// TIA Portal V16 export
// export: Created 2023-03-29T11:04:38.8533234Z, ExportSetting WithDefaults, DisplayName Totally Integrated Automation Portal, DisplayVersion V16 Update 6, DisplayName TIA Portal Version Control Interface, DisplayVersion V16 Update 2, DisplayName TIA Portal Openness, DisplayVersion V16 Update 6, DisplayName STEP 7 Professional, DisplayVersion V16 Update 6, DisplayName STEP 7 Safety, DisplayVersion V16, DisplayName WinCC Advanced, DisplayVersion V16 Update 6
FUNCTION "Read_MPP04_1_ModbusRTU" : Void   // FC23, LAD
TITLE = Read data from SC100
{ S7_Optimized_Access := 'TRUE' }
AUTHOR : rtecmer
VERSION : 0.1
// Czytanie z SC1000 
// Obsługa protokołu Master Modbus RTU.  Odczyt pomiarów  i status czujnika SC1000
// stored: AutoNumber true, IsIECCheckEnabled false, SetENOAutomatically false, UDAEnableTagReadback false
   VAR_TEMP   // added for the SCL form of the ladder/FBD networks
      _w1 : Bool;
      _w2 : Bool;
   END_VAR
BEGIN

REGION Network 1
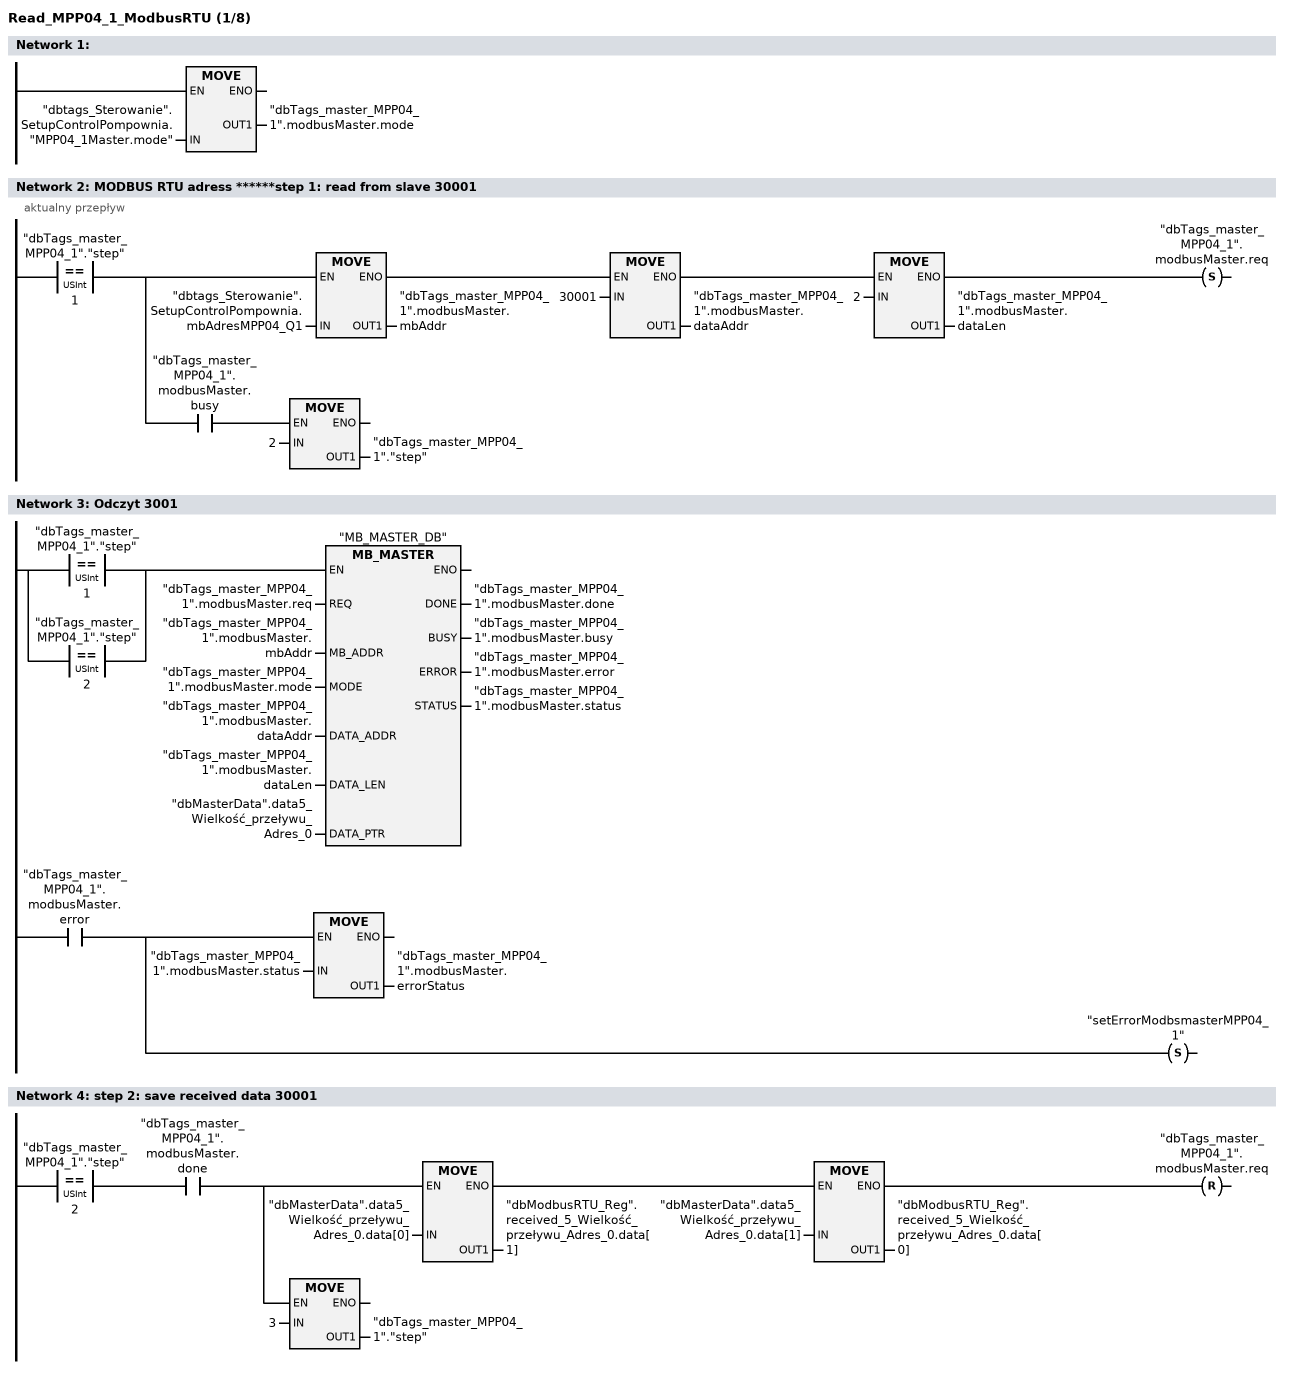
   RUNG wire#powerrail
      { S7_GenerateENO := "TRUE" } Move(in := "dbtags_Sterowanie".SetupControlPompownia."MPP04_1Master.mode", out1 => "dbTags_master_MPP04_1".modbusMaster.mode)
   END_RUNG
   // the same network as SCL:
   "dbTags_master_MPP04_1".modbusMaster.mode := "dbtags_Sterowanie".SetupControlPompownia."MPP04_1Master.mode";
END_REGION

REGION Network 2: MODBUS RTU adress ******step 1: read from slave 30001
   // aktualny przepływ
   RUNG wire#powerrail
      { S7_Templates := "SrcType := USInt" } EQ_Contact(in1 := "dbTags_master_MPP04_1"."step", in2 := 1)
      wire#w1
      Move(in := "dbtags_Sterowanie".SetupControlPompownia.mbAdresMPP04_Q1, out1 => "dbTags_master_MPP04_1".modbusMaster.mbAddr)
      { S7_GenerateENO := "TRUE" } Move(in := 30001, out1 => "dbTags_master_MPP04_1".modbusMaster.dataAddr)
      Move(in := 2, out1 => "dbTags_master_MPP04_1".modbusMaster.dataLen)
      S_Coil( "dbTags_master_MPP04_1".modbusMaster.req )
   END_RUNG
   RUNG wire#w1
      Contact( "dbTags_master_MPP04_1".modbusMaster.busy )
      { S7_GenerateENO := "TRUE" } Move(in := 2, out1 => "dbTags_master_MPP04_1"."step")
   END_RUNG
   // the same network as SCL:
   // ENO of a box is taken as its EN; it also drops when the box reports an error
   #_w1 := "dbTags_master_MPP04_1"."step" = 1;
   IF #_w1 THEN
       "dbTags_master_MPP04_1".modbusMaster.mbAddr := "dbtags_Sterowanie".SetupControlPompownia.mbAdresMPP04_Q1;
       "dbTags_master_MPP04_1".modbusMaster.dataAddr := 30001;
       "dbTags_master_MPP04_1".modbusMaster.dataLen := 2;
       "dbTags_master_MPP04_1".modbusMaster.req := TRUE;
   END_IF;
   IF #_w1 AND "dbTags_master_MPP04_1".modbusMaster.busy THEN "dbTags_master_MPP04_1"."step" := 2; END_IF;
END_REGION

REGION Network 3: Odczyt 3001
   RUNG wire#powerrail
      { S7_Templates := "SrcType := USInt" } EQ_Contact(in1 := "dbTags_master_MPP04_1"."step", in2 := 1)
      wire#w1
      "MB_MASTER_DB".MB_MASTER(REQ := "dbTags_master_MPP04_1".modbusMaster.req, MB_ADDR := "dbTags_master_MPP04_1".modbusMaster.mbAddr, MODE := "dbTags_master_MPP04_1".modbusMaster.mode, DATA_ADDR := "dbTags_master_MPP04_1".modbusMaster.dataAddr, DATA_LEN := "dbTags_master_MPP04_1".modbusMaster.dataLen, DATA_PTR := "dbMasterData".data5_Wielkość_przeływu_Adres_0, DONE => "dbTags_master_MPP04_1".modbusMaster.done, BUSY => "dbTags_master_MPP04_1".modbusMaster.busy, ERROR => "dbTags_master_MPP04_1".modbusMaster.error, STATUS => "dbTags_master_MPP04_1".modbusMaster.status)
   END_RUNG
   RUNG wire#powerrail
      { S7_Templates := "SrcType := USInt" } EQ_Contact(in1 := "dbTags_master_MPP04_1"."step", in2 := 2)
   END_RUNG wire#w1
   RUNG wire#powerrail
      Contact( "dbTags_master_MPP04_1".modbusMaster.error )
      wire#w2
      { S7_GenerateENO := "TRUE" } Move(in := "dbTags_master_MPP04_1".modbusMaster.status, out1 => "dbTags_master_MPP04_1".modbusMaster.errorStatus)
   END_RUNG
   RUNG wire#w2
      S_Coil( "setErrorModbsmasterMPP04_1" )
   END_RUNG
   // the same network as SCL:
   IF ("dbTags_master_MPP04_1"."step" = 1) OR ("dbTags_master_MPP04_1"."step" = 2) THEN
       "MB_MASTER_DB"(REQ := "dbTags_master_MPP04_1".modbusMaster.req,   // MB_MASTER
                      MB_ADDR := "dbTags_master_MPP04_1".modbusMaster.mbAddr,
                      MODE := "dbTags_master_MPP04_1".modbusMaster.mode,
                      DATA_ADDR := "dbTags_master_MPP04_1".modbusMaster.dataAddr,
                      DATA_LEN := "dbTags_master_MPP04_1".modbusMaster.dataLen,
                      DATA_PTR := "dbMasterData".data5_Wielkość_przeływu_Adres_0,
                      DONE => "dbTags_master_MPP04_1".modbusMaster.done,
                      BUSY => "dbTags_master_MPP04_1".modbusMaster.busy,
                      ERROR => "dbTags_master_MPP04_1".modbusMaster.error,
                      STATUS => "dbTags_master_MPP04_1".modbusMaster.status);
   END_IF;
   IF "dbTags_master_MPP04_1".modbusMaster.error THEN
       "dbTags_master_MPP04_1".modbusMaster.errorStatus := "dbTags_master_MPP04_1".modbusMaster.status;
       "setErrorModbsmasterMPP04_1" := TRUE;
   END_IF;
END_REGION

REGION Network 4: step 2: save received data 30001
   RUNG wire#powerrail
      { S7_Templates := "SrcType := USInt" } EQ_Contact(in1 := "dbTags_master_MPP04_1"."step", in2 := 2)
      Contact( "dbTags_master_MPP04_1".modbusMaster.done )
      wire#w1
      { S7_GenerateENO := "TRUE" } Move(in := "dbMasterData".data5_Wielkość_przeływu_Adres_0.data[0], out1 => "dbModbusRTU_Reg".received_5_Wielkość_przeływu_Adres_0.data[1])
      { S7_GenerateENO := "TRUE" } Move(in := "dbMasterData".data5_Wielkość_przeływu_Adres_0.data[1], out1 => "dbModbusRTU_Reg".received_5_Wielkość_przeływu_Adres_0.data[0])
      R_Coil( "dbTags_master_MPP04_1".modbusMaster.req )
   END_RUNG
   RUNG wire#w1
      { S7_GenerateENO := "TRUE" } Move(in := 3, out1 => "dbTags_master_MPP04_1"."step")
   END_RUNG
   // the same network as SCL:
   // ENO of a box is taken as its EN; it also drops when the box reports an error
   IF ("dbTags_master_MPP04_1"."step" = 2) AND "dbTags_master_MPP04_1".modbusMaster.done THEN
       "dbModbusRTU_Reg".received_5_Wielkość_przeływu_Adres_0.data[1] := "dbMasterData".data5_Wielkość_przeływu_Adres_0.data[0];
       "dbModbusRTU_Reg".received_5_Wielkość_przeływu_Adres_0.data[0] := "dbMasterData".data5_Wielkość_przeływu_Adres_0.data[1];
       "dbTags_master_MPP04_1".modbusMaster.req := FALSE;
       "dbTags_master_MPP04_1"."step" := 3;
   END_IF;
END_REGION

REGION Network 5: reakcja na błąd
   // Jęśli błąd pętli modbus lub błąd statusu przepływomierza toustaw 0
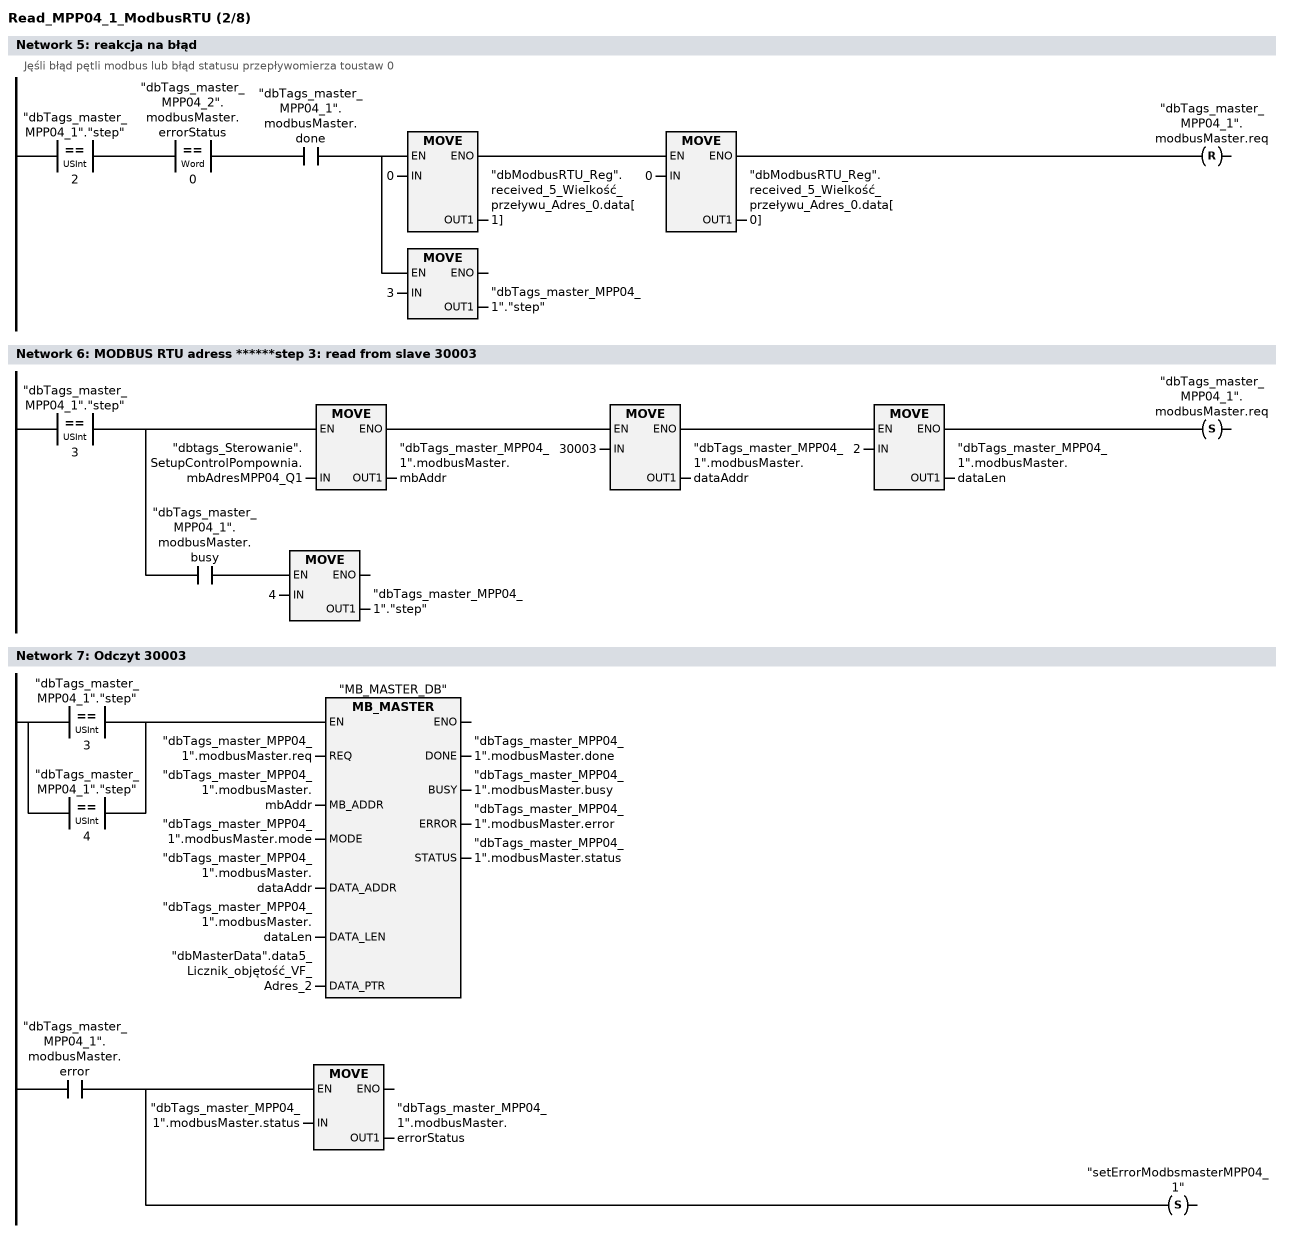
   RUNG wire#powerrail
      { S7_Templates := "SrcType := USInt" } EQ_Contact(in1 := "dbTags_master_MPP04_1"."step", in2 := 2)
      { S7_Templates := "SrcType := Word" } EQ_Contact(in1 := "dbTags_master_MPP04_2".modbusMaster.errorStatus, in2 := 0)
      Contact( "dbTags_master_MPP04_1".modbusMaster.done )
      wire#w1
      { S7_GenerateENO := "TRUE" } Move(in := 0, out1 => "dbModbusRTU_Reg".received_5_Wielkość_przeływu_Adres_0.data[1])
      { S7_GenerateENO := "TRUE" } Move(in := 0, out1 => "dbModbusRTU_Reg".received_5_Wielkość_przeływu_Adres_0.data[0])
      R_Coil( "dbTags_master_MPP04_1".modbusMaster.req )
   END_RUNG
   RUNG wire#w1
      { S7_GenerateENO := "TRUE" } Move(in := 3, out1 => "dbTags_master_MPP04_1"."step")
   END_RUNG
   // the same network as SCL:
   // ENO of a box is taken as its EN; it also drops when the box reports an error
   IF ("dbTags_master_MPP04_1"."step" = 2) AND ("dbTags_master_MPP04_2".modbusMaster.errorStatus = 0) AND "dbTags_master_MPP04_1".modbusMaster.done THEN
       "dbModbusRTU_Reg".received_5_Wielkość_przeływu_Adres_0.data[1] := 0;
       "dbModbusRTU_Reg".received_5_Wielkość_przeływu_Adres_0.data[0] := 0;
       "dbTags_master_MPP04_1".modbusMaster.req := FALSE;
       "dbTags_master_MPP04_1"."step" := 3;
   END_IF;
END_REGION

REGION Network 6: MODBUS RTU adress ******step 3: read from slave 30003
   RUNG wire#powerrail
      { S7_Templates := "SrcType := USInt" } EQ_Contact(in1 := "dbTags_master_MPP04_1"."step", in2 := 3)
      wire#w1
      Move(in := "dbtags_Sterowanie".SetupControlPompownia.mbAdresMPP04_Q1, out1 => "dbTags_master_MPP04_1".modbusMaster.mbAddr)
      { S7_GenerateENO := "TRUE" } Move(in := 30003, out1 => "dbTags_master_MPP04_1".modbusMaster.dataAddr)
      Move(in := 2, out1 => "dbTags_master_MPP04_1".modbusMaster.dataLen)
      S_Coil( "dbTags_master_MPP04_1".modbusMaster.req )
   END_RUNG
   RUNG wire#w1
      Contact( "dbTags_master_MPP04_1".modbusMaster.busy )
      { S7_GenerateENO := "TRUE" } Move(in := 4, out1 => "dbTags_master_MPP04_1"."step")
   END_RUNG
   // the same network as SCL:
   // ENO of a box is taken as its EN; it also drops when the box reports an error
   #_w1 := "dbTags_master_MPP04_1"."step" = 3;
   IF #_w1 THEN
       "dbTags_master_MPP04_1".modbusMaster.mbAddr := "dbtags_Sterowanie".SetupControlPompownia.mbAdresMPP04_Q1;
       "dbTags_master_MPP04_1".modbusMaster.dataAddr := 30003;
       "dbTags_master_MPP04_1".modbusMaster.dataLen := 2;
       "dbTags_master_MPP04_1".modbusMaster.req := TRUE;
   END_IF;
   IF #_w1 AND "dbTags_master_MPP04_1".modbusMaster.busy THEN "dbTags_master_MPP04_1"."step" := 4; END_IF;
END_REGION

REGION Network 7: Odczyt 30003
   RUNG wire#powerrail
      { S7_Templates := "SrcType := USInt" } EQ_Contact(in1 := "dbTags_master_MPP04_1"."step", in2 := 3)
      wire#w1
      "MB_MASTER_DB".MB_MASTER(REQ := "dbTags_master_MPP04_1".modbusMaster.req, MB_ADDR := "dbTags_master_MPP04_1".modbusMaster.mbAddr, MODE := "dbTags_master_MPP04_1".modbusMaster.mode, DATA_ADDR := "dbTags_master_MPP04_1".modbusMaster.dataAddr, DATA_LEN := "dbTags_master_MPP04_1".modbusMaster.dataLen, DATA_PTR := "dbMasterData".data5_Licznik_objętość_VF_Adres_2, DONE => "dbTags_master_MPP04_1".modbusMaster.done, BUSY => "dbTags_master_MPP04_1".modbusMaster.busy, ERROR => "dbTags_master_MPP04_1".modbusMaster.error, STATUS => "dbTags_master_MPP04_1".modbusMaster.status)
   END_RUNG
   RUNG wire#powerrail
      { S7_Templates := "SrcType := USInt" } EQ_Contact(in1 := "dbTags_master_MPP04_1"."step", in2 := 4)
   END_RUNG wire#w1
   RUNG wire#powerrail
      Contact( "dbTags_master_MPP04_1".modbusMaster.error )
      wire#w2
      { S7_GenerateENO := "TRUE" } Move(in := "dbTags_master_MPP04_1".modbusMaster.status, out1 => "dbTags_master_MPP04_1".modbusMaster.errorStatus)
   END_RUNG
   RUNG wire#w2
      S_Coil( "setErrorModbsmasterMPP04_1" )
   END_RUNG
   // the same network as SCL:
   IF ("dbTags_master_MPP04_1"."step" = 3) OR ("dbTags_master_MPP04_1"."step" = 4) THEN
       "MB_MASTER_DB"(REQ := "dbTags_master_MPP04_1".modbusMaster.req,   // MB_MASTER
                      MB_ADDR := "dbTags_master_MPP04_1".modbusMaster.mbAddr,
                      MODE := "dbTags_master_MPP04_1".modbusMaster.mode,
                      DATA_ADDR := "dbTags_master_MPP04_1".modbusMaster.dataAddr,
                      DATA_LEN := "dbTags_master_MPP04_1".modbusMaster.dataLen,
                      DATA_PTR := "dbMasterData".data5_Licznik_objętość_VF_Adres_2,
                      DONE => "dbTags_master_MPP04_1".modbusMaster.done,
                      BUSY => "dbTags_master_MPP04_1".modbusMaster.busy,
                      ERROR => "dbTags_master_MPP04_1".modbusMaster.error,
                      STATUS => "dbTags_master_MPP04_1".modbusMaster.status);
   END_IF;
   IF "dbTags_master_MPP04_1".modbusMaster.error THEN
       "dbTags_master_MPP04_1".modbusMaster.errorStatus := "dbTags_master_MPP04_1".modbusMaster.status;
       "setErrorModbsmasterMPP04_1" := TRUE;
   END_IF;
END_REGION

REGION Network 8: step 4: save received data 30003
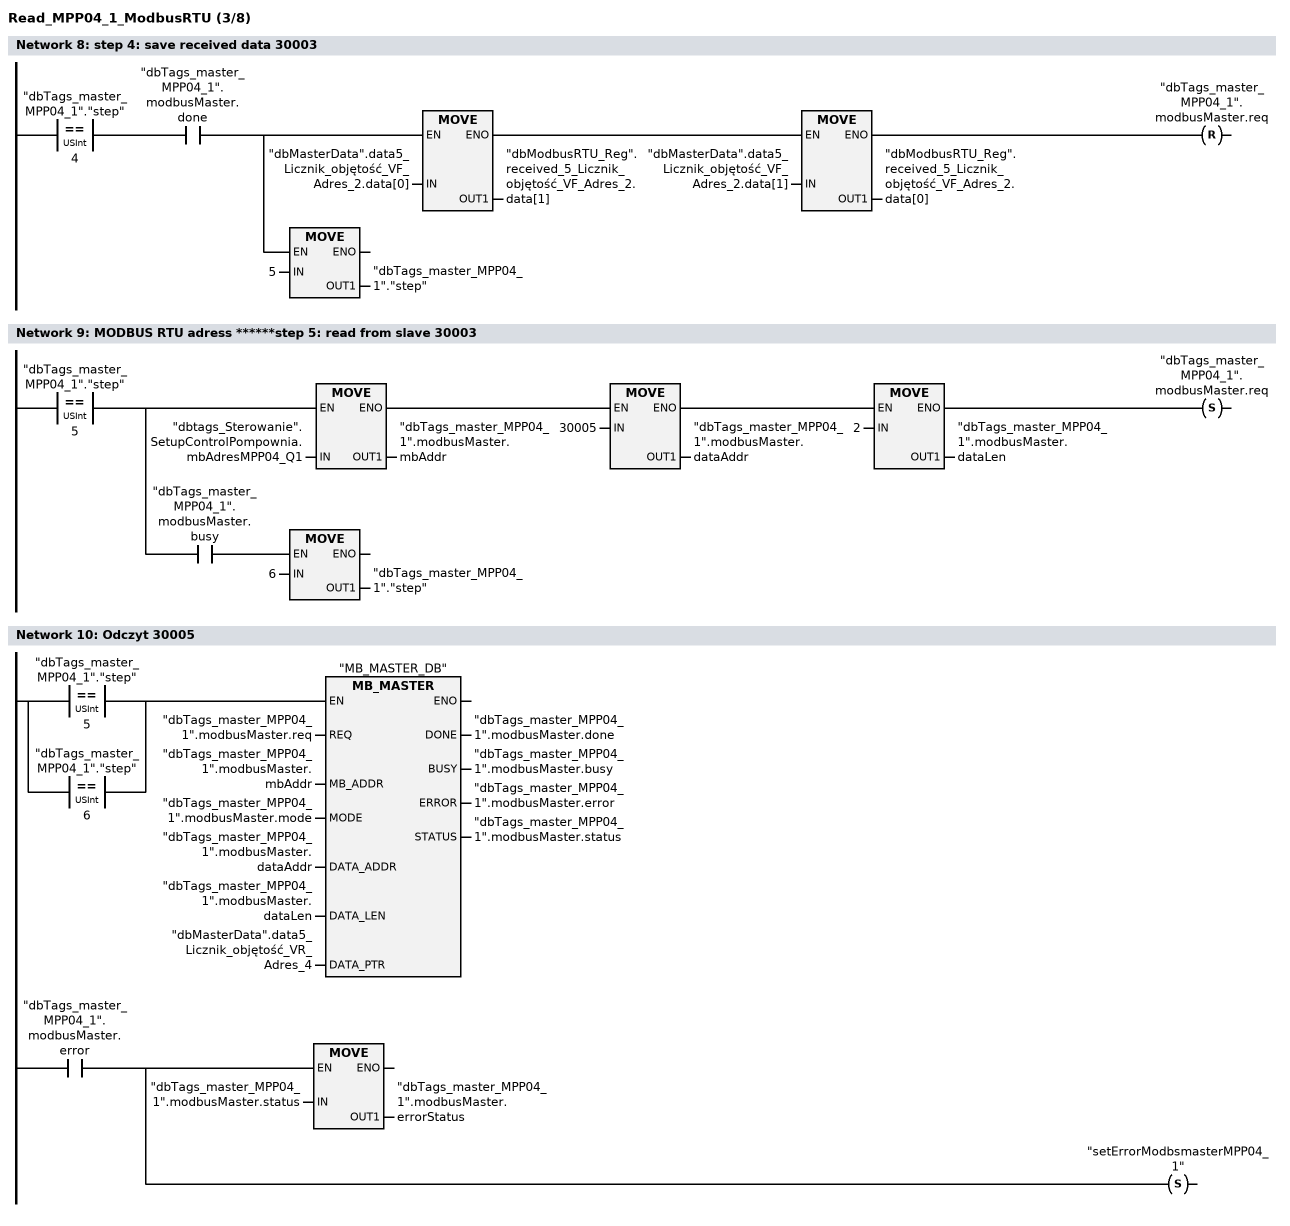
   RUNG wire#powerrail
      { S7_Templates := "SrcType := USInt" } EQ_Contact(in1 := "dbTags_master_MPP04_1"."step", in2 := 4)
      Contact( "dbTags_master_MPP04_1".modbusMaster.done )
      wire#w1
      { S7_GenerateENO := "TRUE" } Move(in := "dbMasterData".data5_Licznik_objętość_VF_Adres_2.data[0], out1 => "dbModbusRTU_Reg".received_5_Licznik_objętość_VF_Adres_2.data[1])
      { S7_GenerateENO := "TRUE" } Move(in := "dbMasterData".data5_Licznik_objętość_VF_Adres_2.data[1], out1 => "dbModbusRTU_Reg".received_5_Licznik_objętość_VF_Adres_2.data[0])
      R_Coil( "dbTags_master_MPP04_1".modbusMaster.req )
   END_RUNG
   RUNG wire#w1
      { S7_GenerateENO := "TRUE" } Move(in := 5, out1 => "dbTags_master_MPP04_1"."step")
   END_RUNG
   // the same network as SCL:
   // ENO of a box is taken as its EN; it also drops when the box reports an error
   IF ("dbTags_master_MPP04_1"."step" = 4) AND "dbTags_master_MPP04_1".modbusMaster.done THEN
       "dbModbusRTU_Reg".received_5_Licznik_objętość_VF_Adres_2.data[1] := "dbMasterData".data5_Licznik_objętość_VF_Adres_2.data[0];
       "dbModbusRTU_Reg".received_5_Licznik_objętość_VF_Adres_2.data[0] := "dbMasterData".data5_Licznik_objętość_VF_Adres_2.data[1];
       "dbTags_master_MPP04_1".modbusMaster.req := FALSE;
       "dbTags_master_MPP04_1"."step" := 5;
   END_IF;
END_REGION

REGION Network 9: MODBUS RTU adress ******step 5: read from slave 30003
   RUNG wire#powerrail
      { S7_Templates := "SrcType := USInt" } EQ_Contact(in1 := "dbTags_master_MPP04_1"."step", in2 := 5)
      wire#w1
      Move(in := "dbtags_Sterowanie".SetupControlPompownia.mbAdresMPP04_Q1, out1 => "dbTags_master_MPP04_1".modbusMaster.mbAddr)
      { S7_GenerateENO := "TRUE" } Move(in := 30005, out1 => "dbTags_master_MPP04_1".modbusMaster.dataAddr)
      Move(in := 2, out1 => "dbTags_master_MPP04_1".modbusMaster.dataLen)
      S_Coil( "dbTags_master_MPP04_1".modbusMaster.req )
   END_RUNG
   RUNG wire#w1
      Contact( "dbTags_master_MPP04_1".modbusMaster.busy )
      { S7_GenerateENO := "TRUE" } Move(in := 6, out1 => "dbTags_master_MPP04_1"."step")
   END_RUNG
   // the same network as SCL:
   // ENO of a box is taken as its EN; it also drops when the box reports an error
   #_w1 := "dbTags_master_MPP04_1"."step" = 5;
   IF #_w1 THEN
       "dbTags_master_MPP04_1".modbusMaster.mbAddr := "dbtags_Sterowanie".SetupControlPompownia.mbAdresMPP04_Q1;
       "dbTags_master_MPP04_1".modbusMaster.dataAddr := 30005;
       "dbTags_master_MPP04_1".modbusMaster.dataLen := 2;
       "dbTags_master_MPP04_1".modbusMaster.req := TRUE;
   END_IF;
   IF #_w1 AND "dbTags_master_MPP04_1".modbusMaster.busy THEN "dbTags_master_MPP04_1"."step" := 6; END_IF;
END_REGION

REGION Network 10: Odczyt 30005
   RUNG wire#powerrail
      { S7_Templates := "SrcType := USInt" } EQ_Contact(in1 := "dbTags_master_MPP04_1"."step", in2 := 5)
      wire#w1
      "MB_MASTER_DB".MB_MASTER(REQ := "dbTags_master_MPP04_1".modbusMaster.req, MB_ADDR := "dbTags_master_MPP04_1".modbusMaster.mbAddr, MODE := "dbTags_master_MPP04_1".modbusMaster.mode, DATA_ADDR := "dbTags_master_MPP04_1".modbusMaster.dataAddr, DATA_LEN := "dbTags_master_MPP04_1".modbusMaster.dataLen, DATA_PTR := "dbMasterData".data5_Licznik_objętość_VR_Adres_4, DONE => "dbTags_master_MPP04_1".modbusMaster.done, BUSY => "dbTags_master_MPP04_1".modbusMaster.busy, ERROR => "dbTags_master_MPP04_1".modbusMaster.error, STATUS => "dbTags_master_MPP04_1".modbusMaster.status)
   END_RUNG
   RUNG wire#powerrail
      { S7_Templates := "SrcType := USInt" } EQ_Contact(in1 := "dbTags_master_MPP04_1"."step", in2 := 6)
   END_RUNG wire#w1
   RUNG wire#powerrail
      Contact( "dbTags_master_MPP04_1".modbusMaster.error )
      wire#w2
      { S7_GenerateENO := "TRUE" } Move(in := "dbTags_master_MPP04_1".modbusMaster.status, out1 => "dbTags_master_MPP04_1".modbusMaster.errorStatus)
   END_RUNG
   RUNG wire#w2
      S_Coil( "setErrorModbsmasterMPP04_1" )
   END_RUNG
   // the same network as SCL:
   IF ("dbTags_master_MPP04_1"."step" = 5) OR ("dbTags_master_MPP04_1"."step" = 6) THEN
       "MB_MASTER_DB"(REQ := "dbTags_master_MPP04_1".modbusMaster.req,   // MB_MASTER
                      MB_ADDR := "dbTags_master_MPP04_1".modbusMaster.mbAddr,
                      MODE := "dbTags_master_MPP04_1".modbusMaster.mode,
                      DATA_ADDR := "dbTags_master_MPP04_1".modbusMaster.dataAddr,
                      DATA_LEN := "dbTags_master_MPP04_1".modbusMaster.dataLen,
                      DATA_PTR := "dbMasterData".data5_Licznik_objętość_VR_Adres_4,
                      DONE => "dbTags_master_MPP04_1".modbusMaster.done,
                      BUSY => "dbTags_master_MPP04_1".modbusMaster.busy,
                      ERROR => "dbTags_master_MPP04_1".modbusMaster.error,
                      STATUS => "dbTags_master_MPP04_1".modbusMaster.status);
   END_IF;
   IF "dbTags_master_MPP04_1".modbusMaster.error THEN
       "dbTags_master_MPP04_1".modbusMaster.errorStatus := "dbTags_master_MPP04_1".modbusMaster.status;
       "setErrorModbsmasterMPP04_1" := TRUE;
   END_IF;
END_REGION

REGION Network 11: step 6: save received data 30005
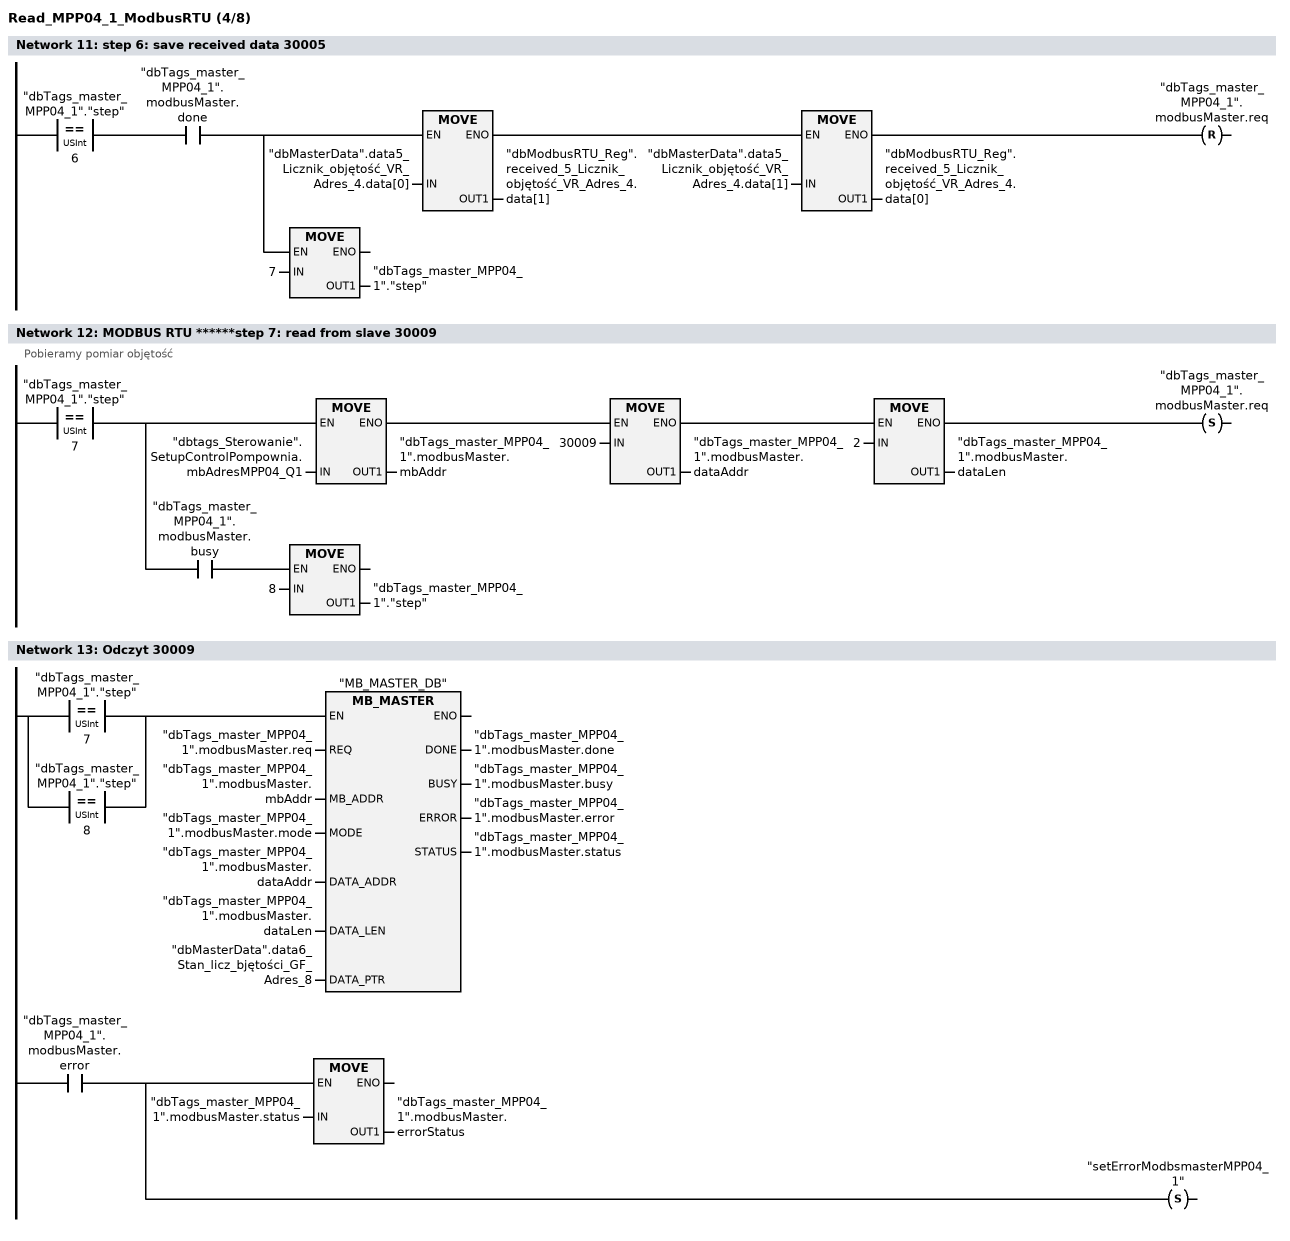
   RUNG wire#powerrail
      { S7_Templates := "SrcType := USInt" } EQ_Contact(in1 := "dbTags_master_MPP04_1"."step", in2 := 6)
      Contact( "dbTags_master_MPP04_1".modbusMaster.done )
      wire#w1
      { S7_GenerateENO := "TRUE" } Move(in := "dbMasterData".data5_Licznik_objętość_VR_Adres_4.data[0], out1 => "dbModbusRTU_Reg".received_5_Licznik_objętość_VR_Adres_4.data[1])
      { S7_GenerateENO := "TRUE" } Move(in := "dbMasterData".data5_Licznik_objętość_VR_Adres_4.data[1], out1 => "dbModbusRTU_Reg".received_5_Licznik_objętość_VR_Adres_4.data[0])
      R_Coil( "dbTags_master_MPP04_1".modbusMaster.req )
   END_RUNG
   RUNG wire#w1
      { S7_GenerateENO := "TRUE" } Move(in := 7, out1 => "dbTags_master_MPP04_1"."step")
   END_RUNG
   // the same network as SCL:
   // ENO of a box is taken as its EN; it also drops when the box reports an error
   IF ("dbTags_master_MPP04_1"."step" = 6) AND "dbTags_master_MPP04_1".modbusMaster.done THEN
       "dbModbusRTU_Reg".received_5_Licznik_objętość_VR_Adres_4.data[1] := "dbMasterData".data5_Licznik_objętość_VR_Adres_4.data[0];
       "dbModbusRTU_Reg".received_5_Licznik_objętość_VR_Adres_4.data[0] := "dbMasterData".data5_Licznik_objętość_VR_Adres_4.data[1];
       "dbTags_master_MPP04_1".modbusMaster.req := FALSE;
       "dbTags_master_MPP04_1"."step" := 7;
   END_IF;
END_REGION

REGION Network 12: MODBUS RTU ******step 7: read from slave 30009
   // Pobieramy pomiar objętość
   RUNG wire#powerrail
      { S7_Templates := "SrcType := USInt" } EQ_Contact(in1 := "dbTags_master_MPP04_1"."step", in2 := 7)
      wire#w1
      Move(in := "dbtags_Sterowanie".SetupControlPompownia.mbAdresMPP04_Q1, out1 => "dbTags_master_MPP04_1".modbusMaster.mbAddr)
      { S7_GenerateENO := "TRUE" } Move(in := 30009, out1 => "dbTags_master_MPP04_1".modbusMaster.dataAddr)
      Move(in := 2, out1 => "dbTags_master_MPP04_1".modbusMaster.dataLen)
      S_Coil( "dbTags_master_MPP04_1".modbusMaster.req )
   END_RUNG
   RUNG wire#w1
      Contact( "dbTags_master_MPP04_1".modbusMaster.busy )
      { S7_GenerateENO := "TRUE" } Move(in := 8, out1 => "dbTags_master_MPP04_1"."step")
   END_RUNG
   // the same network as SCL:
   // ENO of a box is taken as its EN; it also drops when the box reports an error
   #_w1 := "dbTags_master_MPP04_1"."step" = 7;
   IF #_w1 THEN
       "dbTags_master_MPP04_1".modbusMaster.mbAddr := "dbtags_Sterowanie".SetupControlPompownia.mbAdresMPP04_Q1;
       "dbTags_master_MPP04_1".modbusMaster.dataAddr := 30009;
       "dbTags_master_MPP04_1".modbusMaster.dataLen := 2;
       "dbTags_master_MPP04_1".modbusMaster.req := TRUE;
   END_IF;
   IF #_w1 AND "dbTags_master_MPP04_1".modbusMaster.busy THEN "dbTags_master_MPP04_1"."step" := 8; END_IF;
END_REGION

REGION Network 13: Odczyt 30009
   RUNG wire#powerrail
      { S7_Templates := "SrcType := USInt" } EQ_Contact(in1 := "dbTags_master_MPP04_1"."step", in2 := 7)
      wire#w1
      "MB_MASTER_DB".MB_MASTER(REQ := "dbTags_master_MPP04_1".modbusMaster.req, MB_ADDR := "dbTags_master_MPP04_1".modbusMaster.mbAddr, MODE := "dbTags_master_MPP04_1".modbusMaster.mode, DATA_ADDR := "dbTags_master_MPP04_1".modbusMaster.dataAddr, DATA_LEN := "dbTags_master_MPP04_1".modbusMaster.dataLen, DATA_PTR := "dbMasterData".data6_Stan_licz_bjętości_GF_Adres_8, DONE => "dbTags_master_MPP04_1".modbusMaster.done, BUSY => "dbTags_master_MPP04_1".modbusMaster.busy, ERROR => "dbTags_master_MPP04_1".modbusMaster.error, STATUS => "dbTags_master_MPP04_1".modbusMaster.status)
   END_RUNG
   RUNG wire#powerrail
      { S7_Templates := "SrcType := USInt" } EQ_Contact(in1 := "dbTags_master_MPP04_1"."step", in2 := 8)
   END_RUNG wire#w1
   RUNG wire#powerrail
      Contact( "dbTags_master_MPP04_1".modbusMaster.error )
      wire#w2
      { S7_GenerateENO := "TRUE" } Move(in := "dbTags_master_MPP04_1".modbusMaster.status, out1 => "dbTags_master_MPP04_1".modbusMaster.errorStatus)
   END_RUNG
   RUNG wire#w2
      S_Coil( "setErrorModbsmasterMPP04_1" )
   END_RUNG
   // the same network as SCL:
   IF ("dbTags_master_MPP04_1"."step" = 7) OR ("dbTags_master_MPP04_1"."step" = 8) THEN
       "MB_MASTER_DB"(REQ := "dbTags_master_MPP04_1".modbusMaster.req,   // MB_MASTER
                      MB_ADDR := "dbTags_master_MPP04_1".modbusMaster.mbAddr,
                      MODE := "dbTags_master_MPP04_1".modbusMaster.mode,
                      DATA_ADDR := "dbTags_master_MPP04_1".modbusMaster.dataAddr,
                      DATA_LEN := "dbTags_master_MPP04_1".modbusMaster.dataLen,
                      DATA_PTR := "dbMasterData".data6_Stan_licz_bjętości_GF_Adres_8,
                      DONE => "dbTags_master_MPP04_1".modbusMaster.done,
                      BUSY => "dbTags_master_MPP04_1".modbusMaster.busy,
                      ERROR => "dbTags_master_MPP04_1".modbusMaster.error,
                      STATUS => "dbTags_master_MPP04_1".modbusMaster.status);
   END_IF;
   IF "dbTags_master_MPP04_1".modbusMaster.error THEN
       "dbTags_master_MPP04_1".modbusMaster.errorStatus := "dbTags_master_MPP04_1".modbusMaster.status;
       "setErrorModbsmasterMPP04_1" := TRUE;
   END_IF;
END_REGION

REGION Network 14: step 8: save received data 30009
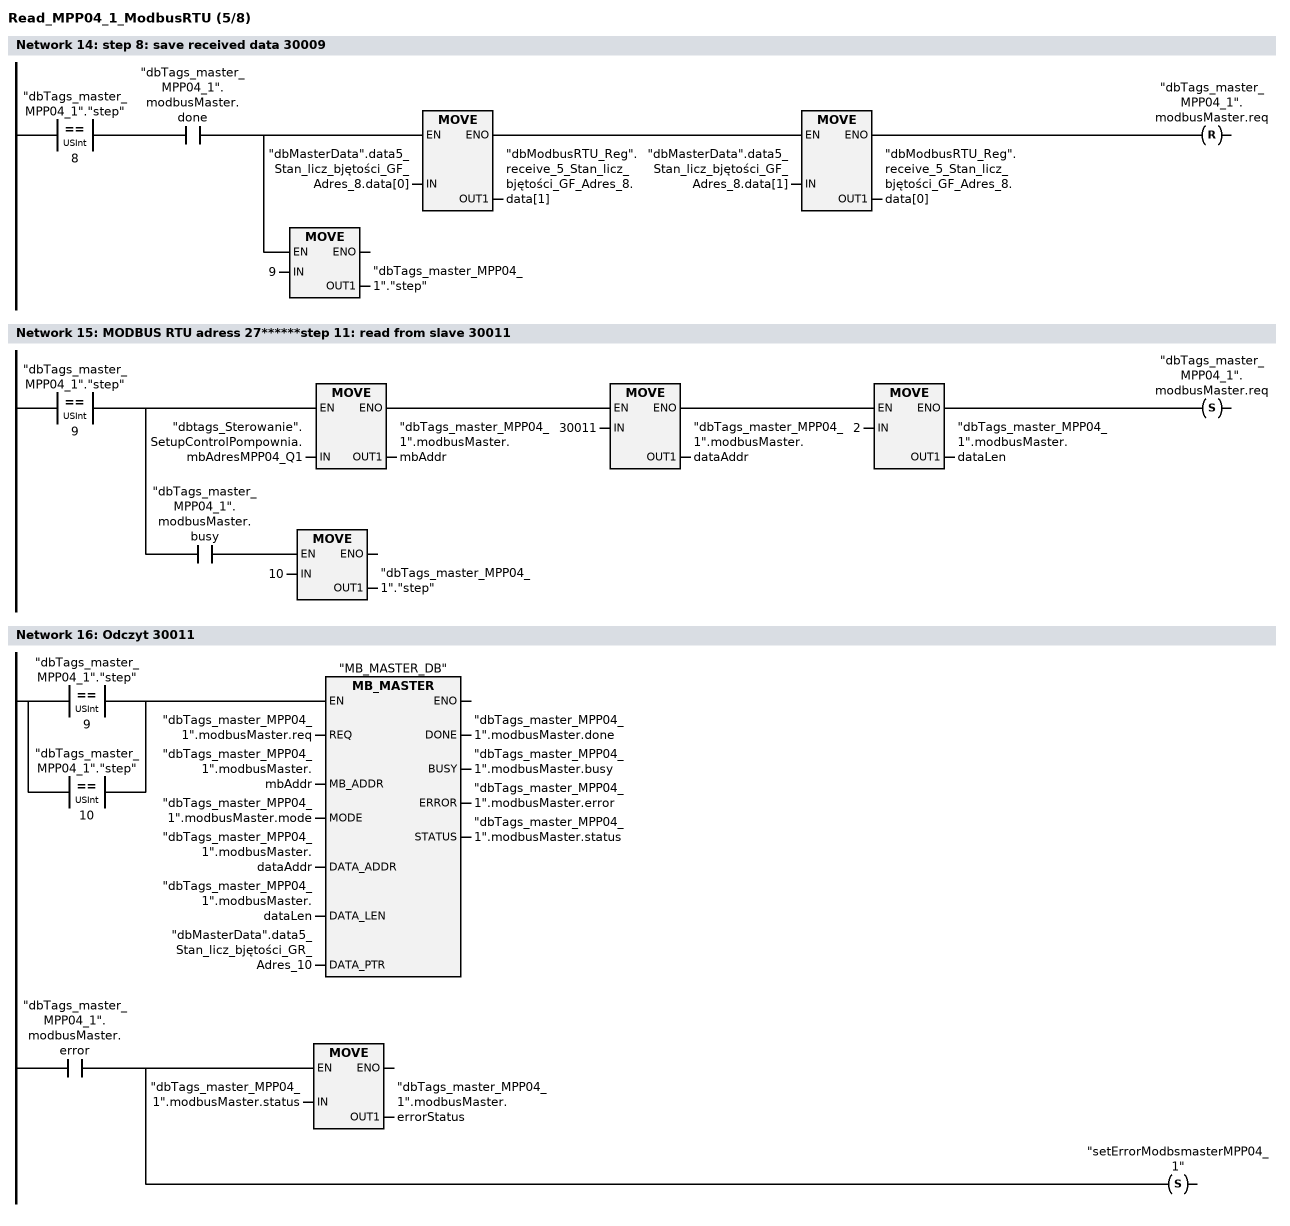
   RUNG wire#powerrail
      { S7_Templates := "SrcType := USInt" } EQ_Contact(in1 := "dbTags_master_MPP04_1"."step", in2 := 8)
      Contact( "dbTags_master_MPP04_1".modbusMaster.done )
      wire#w1
      { S7_GenerateENO := "TRUE" } Move(in := "dbMasterData".data5_Stan_licz_bjętości_GF_Adres_8.data[0], out1 => "dbModbusRTU_Reg".receive_5_Stan_licz_bjętości_GF_Adres_8.data[1])
      { S7_GenerateENO := "TRUE" } Move(in := "dbMasterData".data5_Stan_licz_bjętości_GF_Adres_8.data[1], out1 => "dbModbusRTU_Reg".receive_5_Stan_licz_bjętości_GF_Adres_8.data[0])
      R_Coil( "dbTags_master_MPP04_1".modbusMaster.req )
   END_RUNG
   RUNG wire#w1
      { S7_GenerateENO := "TRUE" } Move(in := 9, out1 => "dbTags_master_MPP04_1"."step")
   END_RUNG
   // the same network as SCL:
   // ENO of a box is taken as its EN; it also drops when the box reports an error
   IF ("dbTags_master_MPP04_1"."step" = 8) AND "dbTags_master_MPP04_1".modbusMaster.done THEN
       "dbModbusRTU_Reg".receive_5_Stan_licz_bjętości_GF_Adres_8.data[1] := "dbMasterData".data5_Stan_licz_bjętości_GF_Adres_8.data[0];
       "dbModbusRTU_Reg".receive_5_Stan_licz_bjętości_GF_Adres_8.data[0] := "dbMasterData".data5_Stan_licz_bjętości_GF_Adres_8.data[1];
       "dbTags_master_MPP04_1".modbusMaster.req := FALSE;
       "dbTags_master_MPP04_1"."step" := 9;
   END_IF;
END_REGION

REGION Network 15: MODBUS RTU adress 27******step 11: read from slave 30011
   RUNG wire#powerrail
      { S7_Templates := "SrcType := USInt" } EQ_Contact(in1 := "dbTags_master_MPP04_1"."step", in2 := 9)
      wire#w1
      Move(in := "dbtags_Sterowanie".SetupControlPompownia.mbAdresMPP04_Q1, out1 => "dbTags_master_MPP04_1".modbusMaster.mbAddr)
      { S7_GenerateENO := "TRUE" } Move(in := 30011, out1 => "dbTags_master_MPP04_1".modbusMaster.dataAddr)
      Move(in := 2, out1 => "dbTags_master_MPP04_1".modbusMaster.dataLen)
      S_Coil( "dbTags_master_MPP04_1".modbusMaster.req )
   END_RUNG
   RUNG wire#w1
      Contact( "dbTags_master_MPP04_1".modbusMaster.busy )
      { S7_GenerateENO := "TRUE" } Move(in := 10, out1 => "dbTags_master_MPP04_1"."step")
   END_RUNG
   // the same network as SCL:
   // ENO of a box is taken as its EN; it also drops when the box reports an error
   #_w1 := "dbTags_master_MPP04_1"."step" = 9;
   IF #_w1 THEN
       "dbTags_master_MPP04_1".modbusMaster.mbAddr := "dbtags_Sterowanie".SetupControlPompownia.mbAdresMPP04_Q1;
       "dbTags_master_MPP04_1".modbusMaster.dataAddr := 30011;
       "dbTags_master_MPP04_1".modbusMaster.dataLen := 2;
       "dbTags_master_MPP04_1".modbusMaster.req := TRUE;
   END_IF;
   IF #_w1 AND "dbTags_master_MPP04_1".modbusMaster.busy THEN "dbTags_master_MPP04_1"."step" := 10; END_IF;
END_REGION

REGION Network 16: Odczyt 30011
   RUNG wire#powerrail
      { S7_Templates := "SrcType := USInt" } EQ_Contact(in1 := "dbTags_master_MPP04_1"."step", in2 := 9)
      wire#w1
      "MB_MASTER_DB".MB_MASTER(REQ := "dbTags_master_MPP04_1".modbusMaster.req, MB_ADDR := "dbTags_master_MPP04_1".modbusMaster.mbAddr, MODE := "dbTags_master_MPP04_1".modbusMaster.mode, DATA_ADDR := "dbTags_master_MPP04_1".modbusMaster.dataAddr, DATA_LEN := "dbTags_master_MPP04_1".modbusMaster.dataLen, DATA_PTR := "dbMasterData".data5_Stan_licz_bjętości_GR_Adres_10, DONE => "dbTags_master_MPP04_1".modbusMaster.done, BUSY => "dbTags_master_MPP04_1".modbusMaster.busy, ERROR => "dbTags_master_MPP04_1".modbusMaster.error, STATUS => "dbTags_master_MPP04_1".modbusMaster.status)
   END_RUNG
   RUNG wire#powerrail
      { S7_Templates := "SrcType := USInt" } EQ_Contact(in1 := "dbTags_master_MPP04_1"."step", in2 := 10)
   END_RUNG wire#w1
   RUNG wire#powerrail
      Contact( "dbTags_master_MPP04_1".modbusMaster.error )
      wire#w2
      { S7_GenerateENO := "TRUE" } Move(in := "dbTags_master_MPP04_1".modbusMaster.status, out1 => "dbTags_master_MPP04_1".modbusMaster.errorStatus)
   END_RUNG
   RUNG wire#w2
      S_Coil( "setErrorModbsmasterMPP04_1" )
   END_RUNG
   // the same network as SCL:
   IF ("dbTags_master_MPP04_1"."step" = 9) OR ("dbTags_master_MPP04_1"."step" = 10) THEN
       "MB_MASTER_DB"(REQ := "dbTags_master_MPP04_1".modbusMaster.req,   // MB_MASTER
                      MB_ADDR := "dbTags_master_MPP04_1".modbusMaster.mbAddr,
                      MODE := "dbTags_master_MPP04_1".modbusMaster.mode,
                      DATA_ADDR := "dbTags_master_MPP04_1".modbusMaster.dataAddr,
                      DATA_LEN := "dbTags_master_MPP04_1".modbusMaster.dataLen,
                      DATA_PTR := "dbMasterData".data5_Stan_licz_bjętości_GR_Adres_10,
                      DONE => "dbTags_master_MPP04_1".modbusMaster.done,
                      BUSY => "dbTags_master_MPP04_1".modbusMaster.busy,
                      ERROR => "dbTags_master_MPP04_1".modbusMaster.error,
                      STATUS => "dbTags_master_MPP04_1".modbusMaster.status);
   END_IF;
   IF "dbTags_master_MPP04_1".modbusMaster.error THEN
       "dbTags_master_MPP04_1".modbusMaster.errorStatus := "dbTags_master_MPP04_1".modbusMaster.status;
       "setErrorModbsmasterMPP04_1" := TRUE;
   END_IF;
END_REGION

REGION Network 17: step 12: save received data 30011
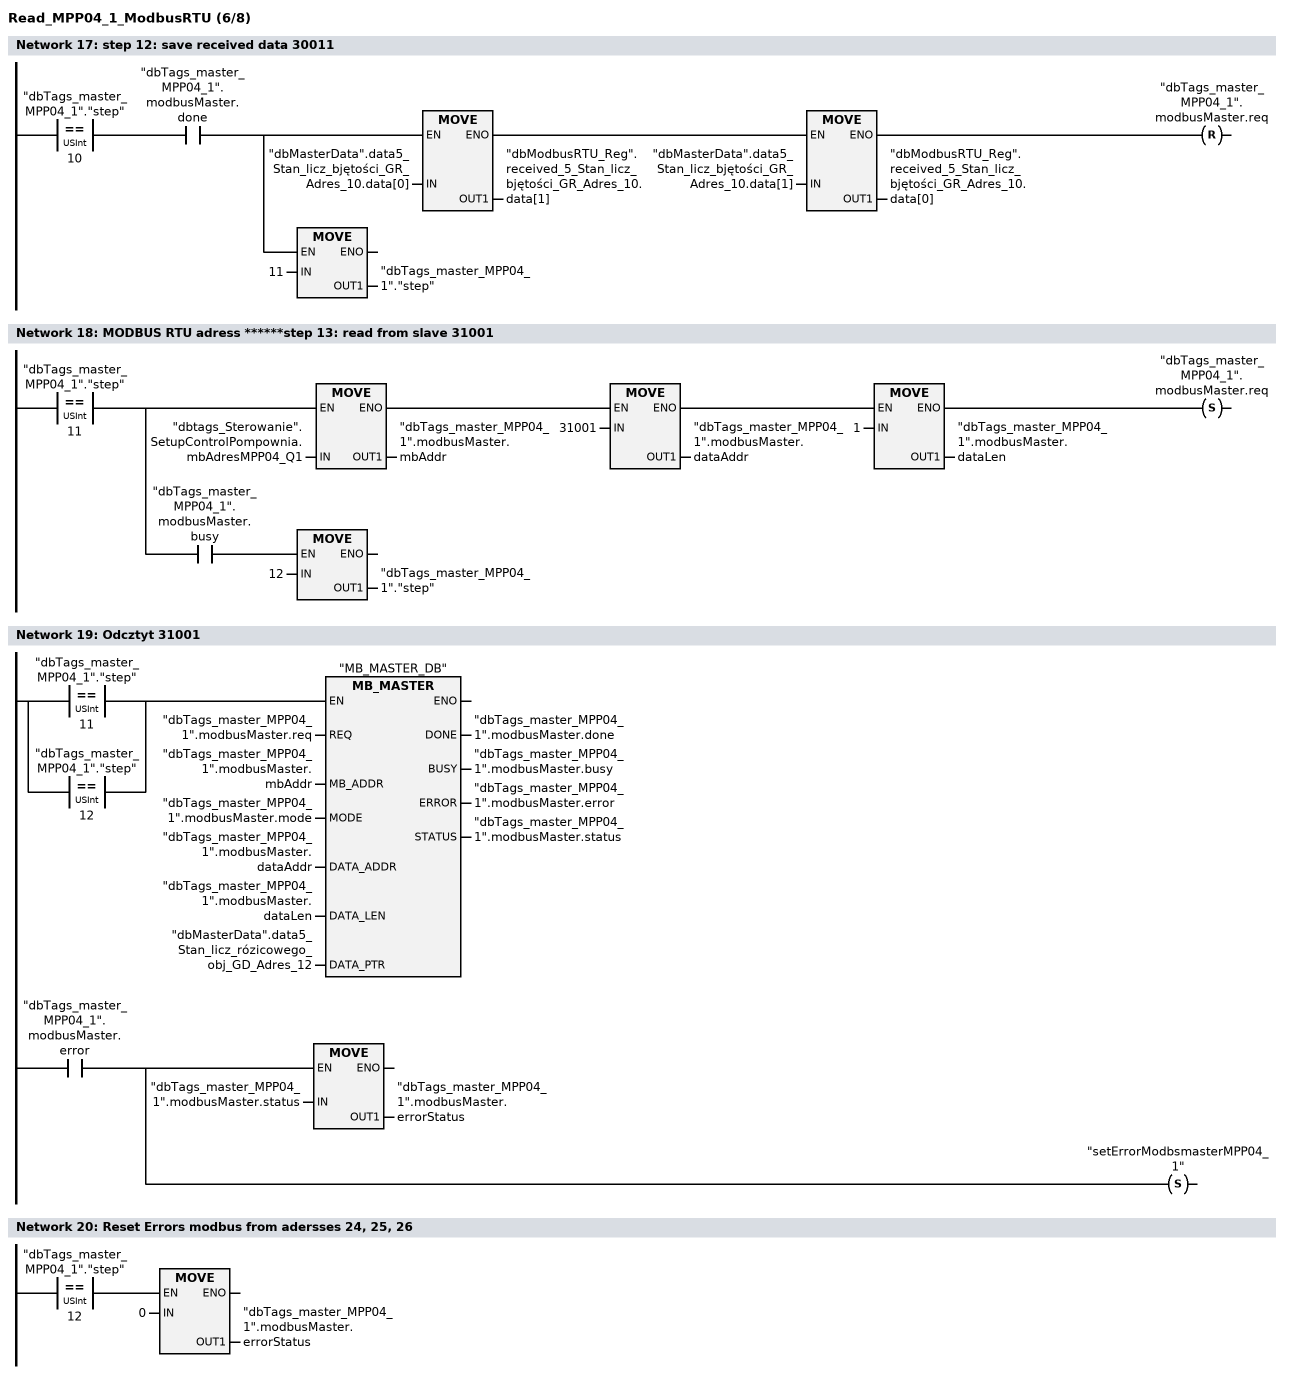
   RUNG wire#powerrail
      { S7_Templates := "SrcType := USInt" } EQ_Contact(in1 := "dbTags_master_MPP04_1"."step", in2 := 10)
      Contact( "dbTags_master_MPP04_1".modbusMaster.done )
      wire#w1
      { S7_GenerateENO := "TRUE" } Move(in := "dbMasterData".data5_Stan_licz_bjętości_GR_Adres_10.data[0], out1 => "dbModbusRTU_Reg".received_5_Stan_licz_bjętości_GR_Adres_10.data[1])
      { S7_GenerateENO := "TRUE" } Move(in := "dbMasterData".data5_Stan_licz_bjętości_GR_Adres_10.data[1], out1 => "dbModbusRTU_Reg".received_5_Stan_licz_bjętości_GR_Adres_10.data[0])
      R_Coil( "dbTags_master_MPP04_1".modbusMaster.req )
   END_RUNG
   RUNG wire#w1
      { S7_GenerateENO := "TRUE" } Move(in := 11, out1 => "dbTags_master_MPP04_1"."step")
   END_RUNG
   // the same network as SCL:
   // ENO of a box is taken as its EN; it also drops when the box reports an error
   IF ("dbTags_master_MPP04_1"."step" = 10) AND "dbTags_master_MPP04_1".modbusMaster.done THEN
       "dbModbusRTU_Reg".received_5_Stan_licz_bjętości_GR_Adres_10.data[1] := "dbMasterData".data5_Stan_licz_bjętości_GR_Adres_10.data[0];
       "dbModbusRTU_Reg".received_5_Stan_licz_bjętości_GR_Adres_10.data[0] := "dbMasterData".data5_Stan_licz_bjętości_GR_Adres_10.data[1];
       "dbTags_master_MPP04_1".modbusMaster.req := FALSE;
       "dbTags_master_MPP04_1"."step" := 11;
   END_IF;
END_REGION

REGION Network 18: MODBUS RTU adress ******step 13: read from slave 31001
   RUNG wire#powerrail
      { S7_Templates := "SrcType := USInt" } EQ_Contact(in1 := "dbTags_master_MPP04_1"."step", in2 := 11)
      wire#w1
      Move(in := "dbtags_Sterowanie".SetupControlPompownia.mbAdresMPP04_Q1, out1 => "dbTags_master_MPP04_1".modbusMaster.mbAddr)
      { S7_GenerateENO := "TRUE" } Move(in := 31001, out1 => "dbTags_master_MPP04_1".modbusMaster.dataAddr)
      Move(in := 1, out1 => "dbTags_master_MPP04_1".modbusMaster.dataLen)
      S_Coil( "dbTags_master_MPP04_1".modbusMaster.req )
   END_RUNG
   RUNG wire#w1
      Contact( "dbTags_master_MPP04_1".modbusMaster.busy )
      { S7_GenerateENO := "TRUE" } Move(in := 12, out1 => "dbTags_master_MPP04_1"."step")
   END_RUNG
   // the same network as SCL:
   // ENO of a box is taken as its EN; it also drops when the box reports an error
   #_w1 := "dbTags_master_MPP04_1"."step" = 11;
   IF #_w1 THEN
       "dbTags_master_MPP04_1".modbusMaster.mbAddr := "dbtags_Sterowanie".SetupControlPompownia.mbAdresMPP04_Q1;
       "dbTags_master_MPP04_1".modbusMaster.dataAddr := 31001;
       "dbTags_master_MPP04_1".modbusMaster.dataLen := 1;
       "dbTags_master_MPP04_1".modbusMaster.req := TRUE;
   END_IF;
   IF #_w1 AND "dbTags_master_MPP04_1".modbusMaster.busy THEN "dbTags_master_MPP04_1"."step" := 12; END_IF;
END_REGION

REGION Network 19: Odcztyt 31001
   RUNG wire#powerrail
      { S7_Templates := "SrcType := USInt" } EQ_Contact(in1 := "dbTags_master_MPP04_1"."step", in2 := 11)
      wire#w1
      "MB_MASTER_DB".MB_MASTER(REQ := "dbTags_master_MPP04_1".modbusMaster.req, MB_ADDR := "dbTags_master_MPP04_1".modbusMaster.mbAddr, MODE := "dbTags_master_MPP04_1".modbusMaster.mode, DATA_ADDR := "dbTags_master_MPP04_1".modbusMaster.dataAddr, DATA_LEN := "dbTags_master_MPP04_1".modbusMaster.dataLen, DATA_PTR := "dbMasterData".data5_Stan_licz_rózicowego_obj_GD_Adres_12, DONE => "dbTags_master_MPP04_1".modbusMaster.done, BUSY => "dbTags_master_MPP04_1".modbusMaster.busy, ERROR => "dbTags_master_MPP04_1".modbusMaster.error, STATUS => "dbTags_master_MPP04_1".modbusMaster.status)
   END_RUNG
   RUNG wire#powerrail
      { S7_Templates := "SrcType := USInt" } EQ_Contact(in1 := "dbTags_master_MPP04_1"."step", in2 := 12)
   END_RUNG wire#w1
   RUNG wire#powerrail
      Contact( "dbTags_master_MPP04_1".modbusMaster.error )
      wire#w2
      { S7_GenerateENO := "TRUE" } Move(in := "dbTags_master_MPP04_1".modbusMaster.status, out1 => "dbTags_master_MPP04_1".modbusMaster.errorStatus)
   END_RUNG
   RUNG wire#w2
      S_Coil( "setErrorModbsmasterMPP04_1" )
   END_RUNG
   // the same network as SCL:
   IF ("dbTags_master_MPP04_1"."step" = 11) OR ("dbTags_master_MPP04_1"."step" = 12) THEN
       "MB_MASTER_DB"(REQ := "dbTags_master_MPP04_1".modbusMaster.req,   // MB_MASTER
                      MB_ADDR := "dbTags_master_MPP04_1".modbusMaster.mbAddr,
                      MODE := "dbTags_master_MPP04_1".modbusMaster.mode,
                      DATA_ADDR := "dbTags_master_MPP04_1".modbusMaster.dataAddr,
                      DATA_LEN := "dbTags_master_MPP04_1".modbusMaster.dataLen,
                      DATA_PTR := "dbMasterData".data5_Stan_licz_rózicowego_obj_GD_Adres_12,
                      DONE => "dbTags_master_MPP04_1".modbusMaster.done,
                      BUSY => "dbTags_master_MPP04_1".modbusMaster.busy,
                      ERROR => "dbTags_master_MPP04_1".modbusMaster.error,
                      STATUS => "dbTags_master_MPP04_1".modbusMaster.status);
   END_IF;
   IF "dbTags_master_MPP04_1".modbusMaster.error THEN
       "dbTags_master_MPP04_1".modbusMaster.errorStatus := "dbTags_master_MPP04_1".modbusMaster.status;
       "setErrorModbsmasterMPP04_1" := TRUE;
   END_IF;
END_REGION

REGION Network 20: Reset Errors modbus from adersses 24, 25, 26
   RUNG wire#powerrail
      { S7_Templates := "SrcType := USInt" } EQ_Contact(in1 := "dbTags_master_MPP04_1"."step", in2 := 12)
      { S7_GenerateENO := "TRUE" } Move(in := 0, out1 => "dbTags_master_MPP04_1".modbusMaster.errorStatus)
   END_RUNG
   // the same network as SCL:
   IF "dbTags_master_MPP04_1"."step" = 12 THEN "dbTags_master_MPP04_1".modbusMaster.errorStatus := 0; END_IF;
END_REGION

REGION Network 21: step 16: save received data 40009
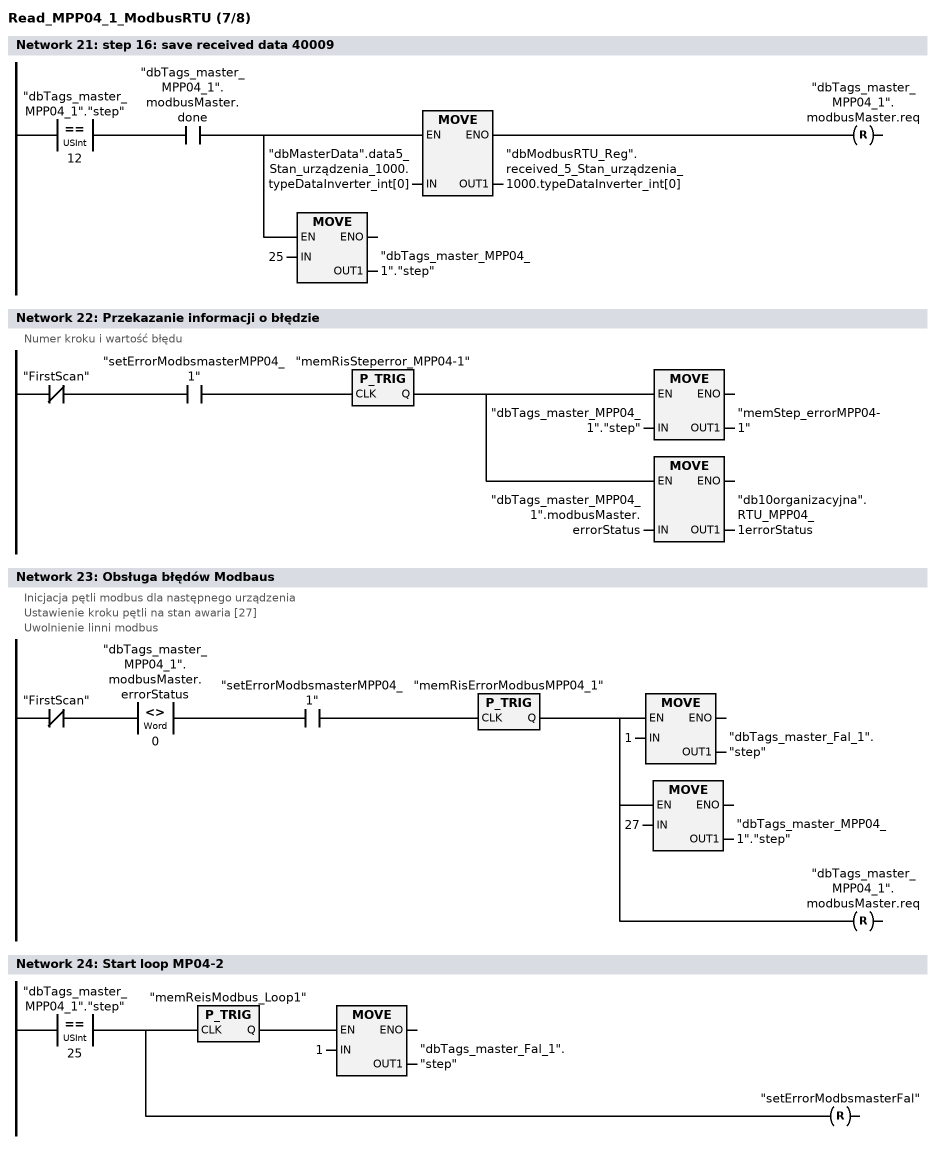
   RUNG wire#powerrail
      { S7_Templates := "SrcType := USInt" } EQ_Contact(in1 := "dbTags_master_MPP04_1"."step", in2 := 12)
      Contact( "dbTags_master_MPP04_1".modbusMaster.done )
      wire#w1
      { S7_GenerateENO := "TRUE" } Move(in := "dbMasterData".data5_Stan_urządzenia_1000.typeDataInverter_int[0], out1 => "dbModbusRTU_Reg".received_5_Stan_urządzenia_1000.typeDataInverter_int[0])
      R_Coil( "dbTags_master_MPP04_1".modbusMaster.req )
   END_RUNG
   RUNG wire#w1
      { S7_GenerateENO := "TRUE" } Move(in := 25, out1 => "dbTags_master_MPP04_1"."step")
   END_RUNG
   // the same network as SCL:
   // ENO of a box is taken as its EN; it also drops when the box reports an error
   IF ("dbTags_master_MPP04_1"."step" = 12) AND "dbTags_master_MPP04_1".modbusMaster.done THEN
       "dbModbusRTU_Reg".received_5_Stan_urządzenia_1000.typeDataInverter_int[0] := "dbMasterData".data5_Stan_urządzenia_1000.typeDataInverter_int[0];
       "dbTags_master_MPP04_1".modbusMaster.req := FALSE;
       "dbTags_master_MPP04_1"."step" := 25;
   END_IF;
END_REGION

REGION Network 22: Przekazanie informacji o błędzie
   // Numer kroku i wartość błędu
   RUNG wire#powerrail
      I_Contact( "FirstScan" )
      Contact( "setErrorModbsmasterMPP04_1" )
      P_Trig( "memRisSteperror_MPP04-1" )
      wire#w1
      Move(in := "dbTags_master_MPP04_1"."step", out1 => "memStep_errorMPP04-1")
   END_RUNG
   RUNG wire#w1
      { S7_GenerateENO := "TRUE" } Move(in := "dbTags_master_MPP04_1".modbusMaster.errorStatus, out1 => "db10organizacyjna".RTU_MPP04_1errorStatus)
   END_RUNG
   // the same network as SCL:
   #_w1 := NOT "FirstScan" AND "setErrorModbsmasterMPP04_1";
   #_w2 := #_w1 AND NOT "memRisSteperror_MPP04-1";   // rising edge
   "memRisSteperror_MPP04-1" := #_w1;
   IF #_w2 THEN
       "memStep_errorMPP04-1" := "dbTags_master_MPP04_1"."step";
       "db10organizacyjna".RTU_MPP04_1errorStatus := "dbTags_master_MPP04_1".modbusMaster.errorStatus;
   END_IF;
END_REGION

REGION Network 23: Obsługa błędów Modbaus
   // Inicjacja pętli modbus dla następnego urządzenia
   // Ustawienie kroku pętli na stan awaria [27]
   // Uwolnienie linni modbus
   RUNG wire#powerrail
      I_Contact( "FirstScan" )
      { S7_Templates := "SrcType := Word" } NE_Contact(in1 := "dbTags_master_MPP04_1".modbusMaster.errorStatus, in2 := 0)
      Contact( "setErrorModbsmasterMPP04_1" )
      P_Trig( "memRisErrorModbusMPP04_1" )
      wire#w1
      { S7_GenerateENO := "TRUE" } Move(in := 1, out1 => "dbTags_master_Fal_1"."step")
   END_RUNG
   RUNG wire#w1
      { S7_GenerateENO := "TRUE" } Move(in := 27, out1 => "dbTags_master_MPP04_1"."step")
   END_RUNG
   RUNG wire#w1
      R_Coil( "dbTags_master_MPP04_1".modbusMaster.req )
   END_RUNG
   // the same network as SCL:
   #_w1 := NOT "FirstScan" AND ("dbTags_master_MPP04_1".modbusMaster.errorStatus <> 0) AND "setErrorModbsmasterMPP04_1";
   #_w2 := #_w1 AND NOT "memRisErrorModbusMPP04_1";   // rising edge
   "memRisErrorModbusMPP04_1" := #_w1;
   IF #_w2 THEN
       "dbTags_master_Fal_1"."step" := 1;
       "dbTags_master_MPP04_1"."step" := 27;
       "dbTags_master_MPP04_1".modbusMaster.req := FALSE;
   END_IF;
END_REGION

REGION Network 24: Start loop MP04-2
   RUNG wire#powerrail
      { S7_Templates := "SrcType := USInt" } EQ_Contact(in1 := "dbTags_master_MPP04_1"."step", in2 := 25)
      wire#w1
      P_Trig( "memReisModbus_Loop1" )
      { S7_GenerateENO := "TRUE" } Move(in := 1, out1 => "dbTags_master_Fal_1"."step")
   END_RUNG
   RUNG wire#w1
      R_Coil( "setErrorModbsmasterFal" )
   END_RUNG
   // the same network as SCL:
   #_w1 := "dbTags_master_MPP04_1"."step" = 25;
   #_w2 := #_w1 AND NOT "memReisModbus_Loop1";   // rising edge
   "memReisModbus_Loop1" := #_w1;
   IF #_w2 THEN "dbTags_master_Fal_1"."step" := 1; END_IF;
   IF #_w1 THEN "setErrorModbsmasterFal" := FALSE; END_IF;
END_REGION

REGION Network 25: Reset error mdbus staus
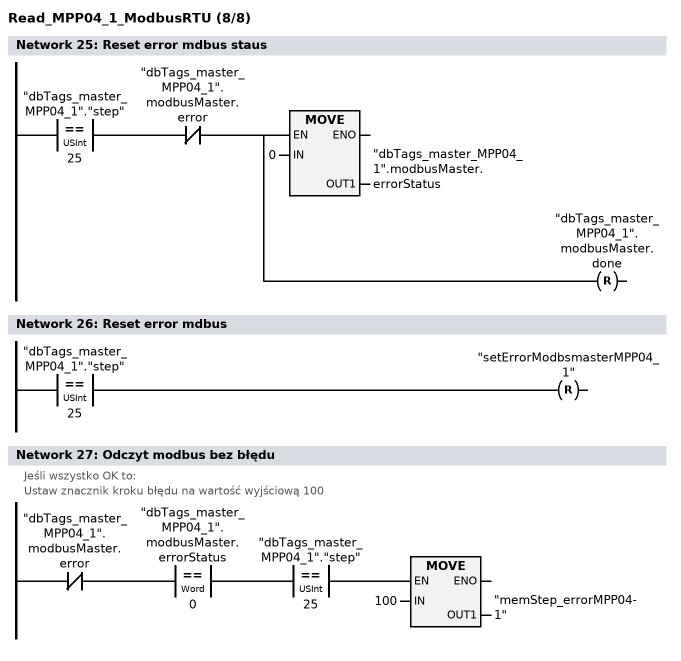
   RUNG wire#powerrail
      { S7_Templates := "SrcType := USInt" } EQ_Contact(in1 := "dbTags_master_MPP04_1"."step", in2 := 25)
      I_Contact( "dbTags_master_MPP04_1".modbusMaster.error )
      wire#w1
      { S7_GenerateENO := "TRUE" } Move(in := 0, out1 => "dbTags_master_MPP04_1".modbusMaster.errorStatus)
   END_RUNG
   RUNG wire#w1
      R_Coil( "dbTags_master_MPP04_1".modbusMaster.done )
   END_RUNG
   // the same network as SCL:
   IF ("dbTags_master_MPP04_1"."step" = 25) AND NOT "dbTags_master_MPP04_1".modbusMaster.error THEN
       "dbTags_master_MPP04_1".modbusMaster.errorStatus := 0;
       "dbTags_master_MPP04_1".modbusMaster.done := FALSE;
   END_IF;
END_REGION

REGION Network 26: Reset error mdbus
   RUNG wire#powerrail
      { S7_Templates := "SrcType := USInt" } EQ_Contact(in1 := "dbTags_master_MPP04_1"."step", in2 := 25)
      R_Coil( "setErrorModbsmasterMPP04_1" )
   END_RUNG
   // the same network as SCL:
   IF "dbTags_master_MPP04_1"."step" = 25 THEN "setErrorModbsmasterMPP04_1" := FALSE; END_IF;
END_REGION

REGION Network 27: Odczyt modbus bez błędu
   // Jeśli wszystko OK to:
   // Ustaw znacznik kroku błędu na wartość wyjściową 100
   RUNG wire#powerrail
      I_Contact( "dbTags_master_MPP04_1".modbusMaster.error )
      { S7_Templates := "SrcType := Word" } EQ_Contact(in1 := "dbTags_master_MPP04_1".modbusMaster.errorStatus, in2 := 0)
      { S7_Templates := "SrcType := USInt" } EQ_Contact(in1 := "dbTags_master_MPP04_1"."step", in2 := 25)
      { S7_GenerateENO := "TRUE" } Move(in := 100, out1 => "memStep_errorMPP04-1")
   END_RUNG
   // the same network as SCL:
   IF NOT "dbTags_master_MPP04_1".modbusMaster.error AND ("dbTags_master_MPP04_1".modbusMaster.errorStatus = 0) AND ("dbTags_master_MPP04_1"."step" = 25) THEN
       "memStep_errorMPP04-1" := 100;
   END_IF;
END_REGION
END_FUNCTION
